(* CODESYS project shid.project

Project tree, tasks and I/O mapping:
  Device : CECC-LK, Festo AG & Co. KG, order no. 574418, version 3.5.7.27
    application Application
      libraries: Standard, * (System); CAA CiA 405, 3.5.0.0 (CAA Technical Workgroup); Solution Center Library, 3.5.8.0 (Festo Didactic SE - Customer Solution Center); OPAK_RFID, 3.5.0.0 (elrest Automationssysteme GmbH); CAA DTUtil Extern, * (CAA Technical Workgroup)
      task MainTask (cyclic, interval t#20ms, priority 20) calls PLC_TO_PC_PROJECT_PRG
      program PLC_PRG [ST]
      program RFID_PRG [ST]
      global variables IO
      program timer_PRG [ST]
      program customTimer_PRG [ST]
      program TCP_PRG [ST]
      program PLC_TO_PC_PROJECT_PRG [ST]
    Onboard : CECC 14I/8O, Festo AG & Co. KG, version 3.4.5.5
        unmapped channels: Onboard Input, Onboard Output
      Digital Inputs
          unmapped channels: Onboard Input
      Digital Outputs
          unmapped channels: Onboard Output
    CAN : CANbus, 3S - Smart Software Solutions GmbH, version 3.5.10.0
        settings: Baudrate = 1000
      CANopen : CANopen_Manager, 3S - Smart Software Solutions GmbH, version 3.5.10.0
          settings: Sync CycleTime in Microseconds = 8000; Synchronous Window Length = 0; Enable Heartbeat generation = FALSE; Factory Settings Default = FALSE; Expert Settings Default = TRUE; ConfigVersion = 50659584
        BL20_GWBR_CANOPEN : BL20-GWBR-CANOPEN, TURCK, order no. 6827167, version Revision=16#00040017, FileVersion=4.23
            settings: General Options.Reset Node = FALSE; NODEIDSAVED = 2; SDO Timeout = 1000000; PDO_Autoconfig = TRUE; EXPERTSETTINGS = TRUE; Emergency-General Parameters.Emergency COBID = 16#00000082; Settings.COBID = 16#00000202; Settings.Transmission Type = 16#FF; Settings.available PDO-Parameter.Inhibit Time available = FALSE; Settings.available PDO-Parameter.Event Timer available = FALSE; Settings.Inhibit Time = 0; Settings.Event Timer = 0; Generic COBID = '$NODEID+16#0200'; Process by CANopenManager = TRUE; Settings.COBID = 16#00000302; Settings.Transmission Type = 16#FF; Settings.available PDO-Parameter.Inhibit Time available = FALSE; Settings.available PDO-Parameter.Event Timer available = FALSE; Settings.Inhibit Time = 0; Settings.Event Timer = 0; Generic COBID = '$NODEID+16#0300'; Process by CANopenManager = TRUE; Settings.COBID = 16#00000182; Settings.Transmission Type = 16#FF; Settings.available PDO-Parameter.Inhibit Time available = TRUE; Settings.available PDO-Parameter.Event Timer available = TRUE; Settings.Inhibit Time = 0; Settings.Event Timer = 0; Generic COBID = '$NODEID+16#0180'; Process by CANopenManager = TRUE; Settings.COBID = 16#00000282; Settings.Transmission Type = 16#FF; Settings.available PDO-Parameter.Inhibit Time available = TRUE; Settings.available PDO-Parameter.Event Timer available = TRUE; Settings.Inhibit Time = 0; Settings.Event Timer = 0; Generic COBID = '$NODEID+16#0280'; Process by CANopenManager = TRUE; WriteOutput8Bit : Generic_BL20_4DO.Index = 16#6200; WriteOutput8Bit : Generic_BL20_4DO.Subindex = 16#01;
              WriteOutput8Bit : Generic_BL20_4DO.ObjectLength = 8; WriteOutput8Bit : Generic_BL20_4DO_2.Index = 16#6200; WriteOutput8Bit : Generic_BL20_4DO_2.Subindex = 16#02; WriteOutput8Bit : Generic_BL20_4DO_2.ObjectLength = 8; WriteAnalogueOutput16 : Generic_BL20_2AO.Index = 16#6411; WriteAnalogueOutput16 : Generic_BL20_2AO.Subindex = 16#01; WriteAnalogueOutput16 : Generic_BL20_2AO.ObjectLength = 16; WriteAnalogueOutput16 : Generic_BL20_2AO.Index = 16#6411; WriteAnalogueOutput16 : Generic_BL20_2AO.Subindex = 16#02; WriteAnalogueOutput16 : Generic_BL20_2AO.ObjectLength = 16; ReadInput8Bit : Generic_BL20_4DI.Index = 16#6000; ReadInput8Bit : Generic_BL20_4DI.Subindex = 16#01; ReadInput8Bit : Generic_BL20_4DI.ObjectLength = 8; ReadAnalogueInput16Bit : Generic_BL20_4AI.Index = 16#6401; ReadAnalogueInput16Bit : Generic_BL20_4AI.Subindex = 16#01; ReadAnalogueInput16Bit : Generic_BL20_4AI.ObjectLength = 16; ReadAnalogueInput16Bit : Generic_BL20_4AI.Index = 16#6401; ReadAnalogueInput16Bit : Generic_BL20_4AI.Subindex = 16#02; ReadAnalogueInput16Bit : Generic_BL20_4AI.ObjectLength = 16; ReadAnalogueInput16Bit : Generic_BL20_4AI.Index = 16#6401; ReadAnalogueInput16Bit : Generic_BL20_4AI.Subindex = 16#03; ReadAnalogueInput16Bit : Generic_BL20_4AI.ObjectLength = 16; ReadAnalogueInput16Bit : Generic_BL20_4AI.Index = 16#6401; ReadAnalogueInput16Bit : Generic_BL20_4AI.Subindex = 16#04; ReadAnalogueInput16Bit : Generic_BL20_4AI.ObjectLength = 16; SDO List.Set Guardtime.Index = 16#100C; SDO List.Set Guardtime.Subindex = 16#00; SDO List.Set Guardtime.Value = 16#00000000; SDO List.Set Guardtime.Size = 16; SDO List.Set Guardtime.AbortIfError = FALSE; SDO List.Set Guardtime.JumpToLine = FALSE; SDO List.Set Guardtime.Line = 0; SDO List.Set Lifetime.Index = 16#100D; SDO List.Set Lifetime.Subindex = 16#00; SDO List.Set Lifetime.Value = 16#00000000; SDO List.Set Lifetime.Size = 8; SDO List.Set Lifetime.AbortIfError = FALSE; SDO List.Set Lifetime.JumpToLine = FALSE; SDO List.Set Lifetime.Line = 0; SDO List.Disable Emcy CobID.Index = 16#1014;
              SDO List.Disable Emcy CobID.Subindex = 16#00; SDO List.Disable Emcy CobID.Value = 16#80000082; SDO List.Disable Emcy CobID.Size = 32; SDO List.Disable Emcy CobID.AbortIfError = FALSE; SDO List.Disable Emcy CobID.JumpToLine = FALSE; SDO List.Disable Emcy CobID.Line = 0; SDO List.Set Emcy CobID.Index = 16#1014; SDO List.Set Emcy CobID.Subindex = 16#00; SDO List.Set Emcy CobID.Value = 16#00000082; SDO List.Set Emcy CobID.Size = 32; SDO List.Set Emcy CobID.AbortIfError = FALSE; SDO List.Set Emcy CobID.JumpToLine = FALSE; SDO List.Set Emcy CobID.Line = 0; SDO List.Set Heartbeat Consumer.Index = 16#1016; SDO List.Set Heartbeat Consumer.Subindex = 16#01; SDO List.Set Heartbeat Consumer.Value = 0; SDO List.Set Heartbeat Consumer.Size = 32; SDO List.Set Heartbeat Consumer.AbortIfError = FALSE; SDO List.Set Heartbeat Consumer.JumpToLine = FALSE; SDO List.Set Heartbeat Consumer.Line = 0; SDO List.Set Heartbeat Producer.Index = 16#1017; SDO List.Set Heartbeat Producer.Subindex = 16#00; SDO List.Set Heartbeat Producer.Value = 16#00000000; SDO List.Set Heartbeat Producer.Size = 16; SDO List.Set Heartbeat Producer.AbortIfError = FALSE; SDO List.Set Heartbeat Producer.JumpToLine = FALSE; SDO List.Set Heartbeat Producer.Line = 0; SDO List.Disable PDO.Index = 16#1400; SDO List.Disable PDO.Subindex = 16#01; SDO List.Disable PDO.Value = 16#80000202; SDO List.Disable PDO.Size = 32; SDO List.Disable PDO.AbortIfError = FALSE; SDO List.Disable PDO.JumpToLine = FALSE; SDO List.Disable PDO.Line = 0; SDO List.Set transmission type.Index = 16#1400; SDO List.Set transmission type.Subindex = 16#02; SDO List.Set transmission type.Value = 16#FF; SDO List.Set transmission type.Size = 8; SDO List.Set transmission type.AbortIfError = FALSE; SDO List.Set transmission type.JumpToLine = FALSE;
              SDO List.Set transmission type.Line = 0; SDO List.Clear pdo mapping.Index = 16#1600; SDO List.Clear pdo mapping.Subindex = 16#00; SDO List.Clear pdo mapping.Value = 16#0; SDO List.Clear pdo mapping.Size = 8; SDO List.Clear pdo mapping.AbortIfError = FALSE; SDO List.Clear pdo mapping.JumpToLine = FALSE; SDO List.Clear pdo mapping.Line = 0; SDO List.Set Mapping.Index = 16#1600; SDO List.Set Mapping.Subindex = 16#01; SDO List.Set Mapping.Value = 16#62000108; SDO List.Set Mapping.Size = 32; SDO List.Set Mapping.AbortIfError = FALSE; SDO List.Set Mapping.JumpToLine = FALSE; SDO List.Set Mapping.Line = 0; SDO List.Set Mapping.Index = 16#1600; SDO List.Set Mapping.Subindex = 16#02; SDO List.Set Mapping.Value = 16#62000208; SDO List.Set Mapping.Size = 32; SDO List.Set Mapping.AbortIfError = FALSE; SDO List.Set Mapping.JumpToLine = FALSE; SDO List.Set Mapping.Line = 0; SDO List.Set number of mappings.Index = 16#1600; SDO List.Set number of mappings.Subindex = 16#00; SDO List.Set number of mappings.Value = 16#02; SDO List.Set number of mappings.Size = 8; SDO List.Set number of mappings.AbortIfError = FALSE; SDO List.Set number of mappings.JumpToLine = FALSE; SDO List.Set number of mappings.Line = 0; SDO List.Set and enable COB-ID.Index = 16#1400; SDO List.Set and enable COB-ID.Subindex = 16#01; SDO List.Set and enable COB-ID.Value = 16#00000202; SDO List.Set and enable COB-ID.Size = 32; SDO List.Set and enable COB-ID.AbortIfError = FALSE; SDO List.Set and enable COB-ID.JumpToLine = FALSE; SDO List.Set and enable COB-ID.Line = 0; SDO List.Disable PDO.Index = 16#1401; SDO List.Disable PDO.Subindex = 16#01; SDO List.Disable PDO.Value = 16#80000302; SDO List.Disable PDO.Size = 32;
              SDO List.Disable PDO.AbortIfError = FALSE; SDO List.Disable PDO.JumpToLine = FALSE; SDO List.Disable PDO.Line = 0; SDO List.Set transmission type.Index = 16#1401; SDO List.Set transmission type.Subindex = 16#02; SDO List.Set transmission type.Value = 16#FF; SDO List.Set transmission type.Size = 8; SDO List.Set transmission type.AbortIfError = FALSE; SDO List.Set transmission type.JumpToLine = FALSE; SDO List.Set transmission type.Line = 0; SDO List.Clear pdo mapping.Index = 16#1601; SDO List.Clear pdo mapping.Subindex = 16#00; SDO List.Clear pdo mapping.Value = 16#0; SDO List.Clear pdo mapping.Size = 8; SDO List.Clear pdo mapping.AbortIfError = FALSE; SDO List.Clear pdo mapping.JumpToLine = FALSE; SDO List.Clear pdo mapping.Line = 0; SDO List.Set Mapping.Index = 16#1601; SDO List.Set Mapping.Subindex = 16#01; SDO List.Set Mapping.Value = 16#64110110; SDO List.Set Mapping.Size = 32; SDO List.Set Mapping.AbortIfError = FALSE; SDO List.Set Mapping.JumpToLine = FALSE; SDO List.Set Mapping.Line = 0; SDO List.Set Mapping.Index = 16#1601; SDO List.Set Mapping.Subindex = 16#02; SDO List.Set Mapping.Value = 16#64110210; SDO List.Set Mapping.Size = 32; SDO List.Set Mapping.AbortIfError = FALSE; SDO List.Set Mapping.JumpToLine = FALSE; SDO List.Set Mapping.Line = 0; SDO List.Set number of mappings.Index = 16#1601; SDO List.Set number of mappings.Subindex = 16#00; SDO List.Set number of mappings.Value = 16#02; SDO List.Set number of mappings.Size = 8; SDO List.Set number of mappings.AbortIfError = FALSE; SDO List.Set number of mappings.JumpToLine = FALSE; SDO List.Set number of mappings.Line = 0; SDO List.Set and enable COB-ID.Index = 16#1401; SDO List.Set and enable COB-ID.Subindex = 16#01;
              SDO List.Set and enable COB-ID.Value = 16#00000302; SDO List.Set and enable COB-ID.Size = 32; SDO List.Set and enable COB-ID.AbortIfError = FALSE; SDO List.Set and enable COB-ID.JumpToLine = FALSE; SDO List.Set and enable COB-ID.Line = 0; SDO List.Disable PDO.Index = 16#1800; SDO List.Disable PDO.Subindex = 16#01; SDO List.Disable PDO.Value = 16#80000182; SDO List.Disable PDO.Size = 32; SDO List.Disable PDO.AbortIfError = FALSE; SDO List.Disable PDO.JumpToLine = FALSE; SDO List.Disable PDO.Line = 0; SDO List.Set transmission type.Index = 16#1800; SDO List.Set transmission type.Subindex = 16#02; SDO List.Set transmission type.Value = 16#FF; SDO List.Set transmission type.Size = 8; SDO List.Set transmission type.AbortIfError = FALSE; SDO List.Set transmission type.JumpToLine = FALSE; SDO List.Set transmission type.Line = 0; SDO List.Set inhibit time.Index = 16#1800; SDO List.Set inhibit time.Subindex = 16#03; SDO List.Set inhibit time.Value = 16#0000; SDO List.Set inhibit time.Size = 16; SDO List.Set inhibit time.AbortIfError = FALSE; SDO List.Set inhibit time.JumpToLine = FALSE; SDO List.Set inhibit time.Line = 0; SDO List.Set event time.Index = 16#1800; SDO List.Set event time.Subindex = 16#05; SDO List.Set event time.Value = 16#0000; SDO List.Set event time.Size = 16; SDO List.Set event time.AbortIfError = FALSE; SDO List.Set event time.JumpToLine = FALSE; SDO List.Set event time.Line = 0; SDO List.Clear pdo mapping.Index = 16#1A00; SDO List.Clear pdo mapping.Subindex = 16#00; SDO List.Clear pdo mapping.Value = 16#0; SDO List.Clear pdo mapping.Size = 8; SDO List.Clear pdo mapping.AbortIfError = FALSE; SDO List.Clear pdo mapping.JumpToLine = FALSE; SDO List.Clear pdo mapping.Line = 0;
              SDO List.Set Mapping.Index = 16#1A00; SDO List.Set Mapping.Subindex = 16#01; SDO List.Set Mapping.Value = 16#60000108; SDO List.Set Mapping.Size = 32; SDO List.Set Mapping.AbortIfError = FALSE; SDO List.Set Mapping.JumpToLine = FALSE; SDO List.Set Mapping.Line = 0; SDO List.Set number of mappings.Index = 16#1A00; SDO List.Set number of mappings.Subindex = 16#00; SDO List.Set number of mappings.Value = 16#01; SDO List.Set number of mappings.Size = 8; SDO List.Set number of mappings.AbortIfError = FALSE; SDO List.Set number of mappings.JumpToLine = FALSE; SDO List.Set number of mappings.Line = 0; SDO List.Set and enable COB-ID.Index = 16#1800; SDO List.Set and enable COB-ID.Subindex = 16#01; SDO List.Set and enable COB-ID.Value = 16#00000182; SDO List.Set and enable COB-ID.Size = 32; SDO List.Set and enable COB-ID.AbortIfError = FALSE; SDO List.Set and enable COB-ID.JumpToLine = FALSE; SDO List.Set and enable COB-ID.Line = 0; SDO List.Disable PDO.Index = 16#1801; SDO List.Disable PDO.Subindex = 16#01; SDO List.Disable PDO.Value = 16#80000282; SDO List.Disable PDO.Size = 32; SDO List.Disable PDO.AbortIfError = FALSE; SDO List.Disable PDO.JumpToLine = FALSE; SDO List.Disable PDO.Line = 0; SDO List.Set transmission type.Index = 16#1801; SDO List.Set transmission type.Subindex = 16#02; SDO List.Set transmission type.Value = 16#FF; SDO List.Set transmission type.Size = 8; SDO List.Set transmission type.AbortIfError = FALSE; SDO List.Set transmission type.JumpToLine = FALSE; SDO List.Set transmission type.Line = 0; SDO List.Set inhibit time.Index = 16#1801; SDO List.Set inhibit time.Subindex = 16#03; SDO List.Set inhibit time.Value = 16#0000; SDO List.Set inhibit time.Size = 16; SDO List.Set inhibit time.AbortIfError = FALSE;
              SDO List.Set inhibit time.JumpToLine = FALSE; SDO List.Set inhibit time.Line = 0; SDO List.Set event time.Index = 16#1801; SDO List.Set event time.Subindex = 16#05; SDO List.Set event time.Value = 16#0000; SDO List.Set event time.Size = 16; SDO List.Set event time.AbortIfError = FALSE; SDO List.Set event time.JumpToLine = FALSE; SDO List.Set event time.Line = 0; SDO List.Clear pdo mapping.Index = 16#1A01; SDO List.Clear pdo mapping.Subindex = 16#00; SDO List.Clear pdo mapping.Value = 16#0; SDO List.Clear pdo mapping.Size = 8; SDO List.Clear pdo mapping.AbortIfError = FALSE; SDO List.Clear pdo mapping.JumpToLine = FALSE; SDO List.Clear pdo mapping.Line = 0; SDO List.Set Mapping.Index = 16#1A01; SDO List.Set Mapping.Subindex = 16#01; SDO List.Set Mapping.Value = 16#64010110; SDO List.Set Mapping.Size = 32; SDO List.Set Mapping.AbortIfError = FALSE; SDO List.Set Mapping.JumpToLine = FALSE; SDO List.Set Mapping.Line = 0; SDO List.Set Mapping.Index = 16#1A01; SDO List.Set Mapping.Subindex = 16#02; SDO List.Set Mapping.Value = 16#64010210; SDO List.Set Mapping.Size = 32; SDO List.Set Mapping.AbortIfError = FALSE; SDO List.Set Mapping.JumpToLine = FALSE; SDO List.Set Mapping.Line = 0; SDO List.Set Mapping.Index = 16#1A01; SDO List.Set Mapping.Subindex = 16#03; SDO List.Set Mapping.Value = 16#64010310; SDO List.Set Mapping.Size = 32; SDO List.Set Mapping.AbortIfError = FALSE; SDO List.Set Mapping.JumpToLine = FALSE; SDO List.Set Mapping.Line = 0; SDO List.Set Mapping.Index = 16#1A01; SDO List.Set Mapping.Subindex = 16#04; SDO List.Set Mapping.Value = 16#64010410;
              SDO List.Set Mapping.Size = 32; SDO List.Set Mapping.AbortIfError = FALSE; SDO List.Set Mapping.JumpToLine = FALSE; SDO List.Set Mapping.Line = 0; SDO List.Set number of mappings.Index = 16#1A01; SDO List.Set number of mappings.Subindex = 16#00; SDO List.Set number of mappings.Value = 16#04; SDO List.Set number of mappings.Size = 8; SDO List.Set number of mappings.AbortIfError = FALSE; SDO List.Set number of mappings.JumpToLine = FALSE; SDO List.Set number of mappings.Line = 0; SDO List.Set and enable COB-ID.Index = 16#1801; SDO List.Set and enable COB-ID.Subindex = 16#01; SDO List.Set and enable COB-ID.Value = 16#00000282; SDO List.Set and enable COB-ID.Size = 32; SDO List.Set and enable COB-ID.AbortIfError = FALSE; SDO List.Set and enable COB-ID.JumpToLine = FALSE; SDO List.Set and enable COB-ID.Line = 0; ConfigVersion = 50659584
          Generic_BL20_4DI : Generic BL20-4DI, TURCK, order no. 0, version Revision=16#00040017, FileVersion=4.23
              settings: Number of Params = 1; ReadInput8Bit : Generic_BL20_4DI.Index = 16#6000; ReadInput8Bit : Generic_BL20_4DI.Subindex = 16#01; ReadInput8Bit : Generic_BL20_4DI.Startbit = 0; ReadInput8Bit : Generic_BL20_4DI.Endbit = 3
              unmapped channels: ReadInput8Bit : Generic_BL20_4DI
          Generic_BL20_4DI_1 : Generic BL20-4DI, TURCK, order no. 0, version Revision=16#00040017, FileVersion=4.23
              settings: Number of Params = 1; ReadInput8Bit : Generic_BL20_4DI.Index = 16#6000; ReadInput8Bit : Generic_BL20_4DI.Subindex = 16#01; ReadInput8Bit : Generic_BL20_4DI.Startbit = 4; ReadInput8Bit : Generic_BL20_4DI.Endbit = 7
              unmapped channels: ReadInput8Bit : Generic_BL20_4DI
          Generic_BL20_BR_PF : Generic BL20-BR/-PF, TURCK, order no. 0, version Revision=16#00040017, FileVersion=4.23
          Generic_BL20_4DO : Generic BL20-4DO, TURCK, order no. 0, version Revision=16#00040017, FileVersion=4.23
              settings: Number of Params = 1; WriteOutput8Bit : Generic_BL20_4DO.Index = 16#6200; WriteOutput8Bit : Generic_BL20_4DO.Subindex = 16#01; WriteOutput8Bit : Generic_BL20_4DO.Startbit = 0; WriteOutput8Bit : Generic_BL20_4DO.Endbit = 3
              unmapped channels: WriteOutput8Bit : Generic_BL20_4DO
          Generic_BL20_4DO_1 : Generic BL20-4DO, TURCK, order no. 0, version Revision=16#00040017, FileVersion=4.23
              settings: Number of Params = 1; WriteOutput8Bit : Generic_BL20_4DO.Index = 16#6200; WriteOutput8Bit : Generic_BL20_4DO.Subindex = 16#01; WriteOutput8Bit : Generic_BL20_4DO.Startbit = 4; WriteOutput8Bit : Generic_BL20_4DO.Endbit = 7
              unmapped channels: WriteOutput8Bit : Generic_BL20_4DO
          Generic_BL20_4DO_2 : Generic BL20-4DO, TURCK, order no. 0, version Revision=16#00040017, FileVersion=4.23
              settings: Number of Params = 1; WriteOutput8Bit : Generic_BL20_4DO_2.Index = 16#6200; WriteOutput8Bit : Generic_BL20_4DO_2.Subindex = 16#02; WriteOutput8Bit : Generic_BL20_4DO_2.Startbit = 0; WriteOutput8Bit : Generic_BL20_4DO_2.Endbit = 3
              unmapped channels: WriteOutput8Bit : Generic_BL20_4DO_2
          Generic_BL20_4DO_3 : Generic BL20-4DO, TURCK, order no. 0, version Revision=16#00040017, FileVersion=4.23
              settings: Number of Params = 1; WriteOutput8Bit : Generic_BL20_4DO_2.Index = 16#6200; WriteOutput8Bit : Generic_BL20_4DO_2.Subindex = 16#02; WriteOutput8Bit : Generic_BL20_4DO_2.Startbit = 4; WriteOutput8Bit : Generic_BL20_4DO_2.Endbit = 7
              unmapped channels: WriteOutput8Bit : Generic_BL20_4DO_2
          Generic_BL20_4AI : Generic BL20-4AI, TURCK, order no. 0, version Revision=16#00040017, FileVersion=4.23
              settings: Number of Params = 4; ReadAnalogueInput16Bit : Generic_BL20_4AI.Index = 16#6401; ReadAnalogueInput16Bit : Generic_BL20_4AI.Subindex = 16#01; ReadAnalogueInput16Bit : Generic_BL20_4AI.Startbit = 0; ReadAnalogueInput16Bit : Generic_BL20_4AI.Endbit = 15; ReadAnalogueInput16Bit : Generic_BL20_4AI.Index = 16#6401; ReadAnalogueInput16Bit : Generic_BL20_4AI.Subindex = 16#02; ReadAnalogueInput16Bit : Generic_BL20_4AI.Startbit = 0; ReadAnalogueInput16Bit : Generic_BL20_4AI.Endbit = 15; ReadAnalogueInput16Bit : Generic_BL20_4AI.Index = 16#6401; ReadAnalogueInput16Bit : Generic_BL20_4AI.Subindex = 16#03; ReadAnalogueInput16Bit : Generic_BL20_4AI.Startbit = 0; ReadAnalogueInput16Bit : Generic_BL20_4AI.Endbit = 15; ReadAnalogueInput16Bit : Generic_BL20_4AI.Index = 16#6401; ReadAnalogueInput16Bit : Generic_BL20_4AI.Subindex = 16#04; ReadAnalogueInput16Bit : Generic_BL20_4AI.Startbit = 0; ReadAnalogueInput16Bit : Generic_BL20_4AI.Endbit = 15
              unmapped channels: ReadAnalogueInput16Bit : Generic_BL20_4AI, ReadAnalogueInput16Bit : Generic_BL20_4AI, ReadAnalogueInput16Bit : Generic_BL20_4AI, ReadAnalogueInput16Bit : Generic_BL20_4AI
          Generic_BL20_2AO : Generic BL20-2AO, TURCK, order no. 0, version Revision=16#00040017, FileVersion=4.23
              settings: Number of Params = 2; WriteAnalogueOutput16 : Generic_BL20_2AO.Index = 16#6411; WriteAnalogueOutput16 : Generic_BL20_2AO.Subindex = 16#01; WriteAnalogueOutput16 : Generic_BL20_2AO.Startbit = 0; WriteAnalogueOutput16 : Generic_BL20_2AO.Endbit = 15; WriteAnalogueOutput16 : Generic_BL20_2AO.Index = 16#6411; WriteAnalogueOutput16 : Generic_BL20_2AO.Subindex = 16#02; WriteAnalogueOutput16 : Generic_BL20_2AO.Startbit = 0; WriteAnalogueOutput16 : Generic_BL20_2AO.Endbit = 15
              unmapped channels: WriteAnalogueOutput16 : Generic_BL20_2AO, WriteAnalogueOutput16 : Generic_BL20_2AO
        DTM425 : DTM425, ifm electronic gmbh, order no. DTM425, version Revision=16#00000000, FileVersion=8.2, File=DTM425.eds
            settings: General Options.Reset Node = FALSE; NODEIDSAVED = 32; SDO Timeout = 1000000; PDO_Autoconfig = FALSE; EXPERTSETTINGS = TRUE; Emergency-General Parameters.Emergency COBID = 16#000000A0; PDO 16#1400.COBID = 16#00000220; Process by CANopenManager = TRUE; PDO 16#1401.COBID = 16#00000320; Process by CANopenManager = TRUE; PDO 16#1402.COBID = 16#00000420; Process by CANopenManager = TRUE; PDO 16#1403.COBID = 16#00000520; Process by CANopenManager = TRUE; PDO 16#1800.COBID = 16#000001A0; PDO 16#1800.Event Timer = 0; Process by CANopenManager = TRUE; PDO 16#1801.COBID = 16#000002A0; PDO 16#1801.Event Timer = 0; Process by CANopenManager = TRUE; PDO 16#1802.COBID = 16#000003A0; PDO 16#1802.Event Timer = 0; Process by CANopenManager = TRUE; PDO 16#1803.COBID = 16#000004A0; PDO 16#1803.Event Timer = 0; Process by CANopenManager = TRUE; Write Data (mappable): Write Trigger.Subindex = 16#00; Write Data (mappable): Data_sub1.Subindex = 16#01; Write Data (mappable): Data_sub2.Subindex = 16#02; Write Data (mappable): Data_sub3.Subindex = 16#03; Device Status.Subindex = 16#00; Read Data (mappable): Data_sub1.Subindex = 16#01; Read Data (mappable): Data_sub2.Subindex = 16#02; Read Data (mappable): Data_sub3.Subindex = 16#03; SDO List.Disable Emcy CobID.Index = 16#1014; SDO List.Disable Emcy CobID.Subindex = 16#00; SDO List.Disable Emcy CobID.Value = 16#800000A0; SDO List.Disable Emcy CobID.Size = 32; SDO List.Disable Emcy CobID.AbortIfError = FALSE; SDO List.Disable Emcy CobID.JumpToLine = FALSE;
              SDO List.Disable Emcy CobID.Line = 0; SDO List.Set Emcy CobID.Index = 16#1014; SDO List.Set Emcy CobID.Subindex = 16#00; SDO List.Set Emcy CobID.Value = 16#000000A0; SDO List.Set Emcy CobID.Size = 32; SDO List.Set Emcy CobID.AbortIfError = FALSE; SDO List.Set Emcy CobID.JumpToLine = FALSE; SDO List.Set Emcy CobID.Line = 0; SDO List.Set Heartbeat Producer.Index = 16#1017; SDO List.Set Heartbeat Producer.Subindex = 16#00; SDO List.Set Heartbeat Producer.Value = 16#00000000; SDO List.Set Heartbeat Producer.Size = 16; SDO List.Set Heartbeat Producer.AbortIfError = FALSE; SDO List.Set Heartbeat Producer.JumpToLine = FALSE; SDO List.Set Heartbeat Producer.Line = 0; SDO List.Disable PDO.Index = 16#1400; SDO List.Disable PDO.Subindex = 16#01; SDO List.Disable PDO.Value = 16#80000220; SDO List.Disable PDO.Size = 32; SDO List.Disable PDO.AbortIfError = FALSE; SDO List.Disable PDO.JumpToLine = FALSE; SDO List.Disable PDO.Line = 0; SDO List.Set transmission type.Index = 16#1400; SDO List.Set transmission type.Subindex = 16#02; SDO List.Set transmission type.Value = 16#FF; SDO List.Set transmission type.Size = 8; SDO List.Set transmission type.AbortIfError = FALSE; SDO List.Set transmission type.JumpToLine = FALSE; SDO List.Set transmission type.Line = 0; SDO List.Clear pdo mapping.Index = 16#1600; SDO List.Clear pdo mapping.Subindex = 16#00; SDO List.Clear pdo mapping.Value = 16#0; SDO List.Clear pdo mapping.Size = 8; SDO List.Clear pdo mapping.AbortIfError = FALSE; SDO List.Clear pdo mapping.JumpToLine = FALSE; SDO List.Clear pdo mapping.Line = 0; SDO List.Set Mapping.Index = 16#1600; SDO List.Set Mapping.Subindex = 16#01; SDO List.Set Mapping.Value = 16#230F0040; SDO List.Set Mapping.Size = 32;
              SDO List.Set Mapping.AbortIfError = FALSE; SDO List.Set Mapping.JumpToLine = FALSE; SDO List.Set Mapping.Line = 0; SDO List.Set number of mappings.Index = 16#1600; SDO List.Set number of mappings.Subindex = 16#00; SDO List.Set number of mappings.Value = 16#01; SDO List.Set number of mappings.Size = 8; SDO List.Set number of mappings.AbortIfError = FALSE; SDO List.Set number of mappings.JumpToLine = FALSE; SDO List.Set number of mappings.Line = 0; SDO List.Set and enable COB-ID.Index = 16#1400; SDO List.Set and enable COB-ID.Subindex = 16#01; SDO List.Set and enable COB-ID.Value = 16#00000220; SDO List.Set and enable COB-ID.Size = 32; SDO List.Set and enable COB-ID.AbortIfError = FALSE; SDO List.Set and enable COB-ID.JumpToLine = FALSE; SDO List.Set and enable COB-ID.Line = 0; SDO List.Disable PDO.Index = 16#1401; SDO List.Disable PDO.Subindex = 16#01; SDO List.Disable PDO.Value = 16#80000320; SDO List.Disable PDO.Size = 32; SDO List.Disable PDO.AbortIfError = FALSE; SDO List.Disable PDO.JumpToLine = FALSE; SDO List.Disable PDO.Line = 0; SDO List.Set transmission type.Index = 16#1401; SDO List.Set transmission type.Subindex = 16#02; SDO List.Set transmission type.Value = 16#FF; SDO List.Set transmission type.Size = 8; SDO List.Set transmission type.AbortIfError = FALSE; SDO List.Set transmission type.JumpToLine = FALSE; SDO List.Set transmission type.Line = 0; SDO List.Clear pdo mapping.Index = 16#1601; SDO List.Clear pdo mapping.Subindex = 16#00; SDO List.Clear pdo mapping.Value = 16#0; SDO List.Clear pdo mapping.Size = 8; SDO List.Clear pdo mapping.AbortIfError = FALSE; SDO List.Clear pdo mapping.JumpToLine = FALSE; SDO List.Clear pdo mapping.Line = 0; SDO List.Set Mapping.Index = 16#1601; SDO List.Set Mapping.Subindex = 16#01;
              SDO List.Set Mapping.Value = 16#230A0140; SDO List.Set Mapping.Size = 32; SDO List.Set Mapping.AbortIfError = FALSE; SDO List.Set Mapping.JumpToLine = FALSE; SDO List.Set Mapping.Line = 0; SDO List.Set number of mappings.Index = 16#1601; SDO List.Set number of mappings.Subindex = 16#00; SDO List.Set number of mappings.Value = 16#01; SDO List.Set number of mappings.Size = 8; SDO List.Set number of mappings.AbortIfError = FALSE; SDO List.Set number of mappings.JumpToLine = FALSE; SDO List.Set number of mappings.Line = 0; SDO List.Set and enable COB-ID.Index = 16#1401; SDO List.Set and enable COB-ID.Subindex = 16#01; SDO List.Set and enable COB-ID.Value = 16#00000320; SDO List.Set and enable COB-ID.Size = 32; SDO List.Set and enable COB-ID.AbortIfError = FALSE; SDO List.Set and enable COB-ID.JumpToLine = FALSE; SDO List.Set and enable COB-ID.Line = 0; SDO List.Disable PDO.Index = 16#1402; SDO List.Disable PDO.Subindex = 16#01; SDO List.Disable PDO.Value = 16#80000420; SDO List.Disable PDO.Size = 32; SDO List.Disable PDO.AbortIfError = FALSE; SDO List.Disable PDO.JumpToLine = FALSE; SDO List.Disable PDO.Line = 0; SDO List.Set transmission type.Index = 16#1402; SDO List.Set transmission type.Subindex = 16#02; SDO List.Set transmission type.Value = 16#FF; SDO List.Set transmission type.Size = 8; SDO List.Set transmission type.AbortIfError = FALSE; SDO List.Set transmission type.JumpToLine = FALSE; SDO List.Set transmission type.Line = 0; SDO List.Clear pdo mapping.Index = 16#1602; SDO List.Clear pdo mapping.Subindex = 16#00; SDO List.Clear pdo mapping.Value = 16#0; SDO List.Clear pdo mapping.Size = 8; SDO List.Clear pdo mapping.AbortIfError = FALSE; SDO List.Clear pdo mapping.JumpToLine = FALSE; SDO List.Clear pdo mapping.Line = 0;
              SDO List.Set Mapping.Index = 16#1602; SDO List.Set Mapping.Subindex = 16#01; SDO List.Set Mapping.Value = 16#230A0240; SDO List.Set Mapping.Size = 32; SDO List.Set Mapping.AbortIfError = FALSE; SDO List.Set Mapping.JumpToLine = FALSE; SDO List.Set Mapping.Line = 0; SDO List.Set number of mappings.Index = 16#1602; SDO List.Set number of mappings.Subindex = 16#00; SDO List.Set number of mappings.Value = 16#01; SDO List.Set number of mappings.Size = 8; SDO List.Set number of mappings.AbortIfError = FALSE; SDO List.Set number of mappings.JumpToLine = FALSE; SDO List.Set number of mappings.Line = 0; SDO List.Set and enable COB-ID.Index = 16#1402; SDO List.Set and enable COB-ID.Subindex = 16#01; SDO List.Set and enable COB-ID.Value = 16#00000420; SDO List.Set and enable COB-ID.Size = 32; SDO List.Set and enable COB-ID.AbortIfError = FALSE; SDO List.Set and enable COB-ID.JumpToLine = FALSE; SDO List.Set and enable COB-ID.Line = 0; SDO List.Disable PDO.Index = 16#1403; SDO List.Disable PDO.Subindex = 16#01; SDO List.Disable PDO.Value = 16#80000520; SDO List.Disable PDO.Size = 32; SDO List.Disable PDO.AbortIfError = FALSE; SDO List.Disable PDO.JumpToLine = FALSE; SDO List.Disable PDO.Line = 0; SDO List.Set transmission type.Index = 16#1403; SDO List.Set transmission type.Subindex = 16#02; SDO List.Set transmission type.Value = 16#FF; SDO List.Set transmission type.Size = 8; SDO List.Set transmission type.AbortIfError = FALSE; SDO List.Set transmission type.JumpToLine = FALSE; SDO List.Set transmission type.Line = 0; SDO List.Clear pdo mapping.Index = 16#1603; SDO List.Clear pdo mapping.Subindex = 16#00; SDO List.Clear pdo mapping.Value = 16#0; SDO List.Clear pdo mapping.Size = 8; SDO List.Clear pdo mapping.AbortIfError = FALSE;
              SDO List.Clear pdo mapping.JumpToLine = FALSE; SDO List.Clear pdo mapping.Line = 0; SDO List.Set Mapping.Index = 16#1603; SDO List.Set Mapping.Subindex = 16#01; SDO List.Set Mapping.Value = 16#230A0340; SDO List.Set Mapping.Size = 32; SDO List.Set Mapping.AbortIfError = FALSE; SDO List.Set Mapping.JumpToLine = FALSE; SDO List.Set Mapping.Line = 0; SDO List.Set number of mappings.Index = 16#1603; SDO List.Set number of mappings.Subindex = 16#00; SDO List.Set number of mappings.Value = 16#01; SDO List.Set number of mappings.Size = 8; SDO List.Set number of mappings.AbortIfError = FALSE; SDO List.Set number of mappings.JumpToLine = FALSE; SDO List.Set number of mappings.Line = 0; SDO List.Set and enable COB-ID.Index = 16#1403; SDO List.Set and enable COB-ID.Subindex = 16#01; SDO List.Set and enable COB-ID.Value = 16#00000520; SDO List.Set and enable COB-ID.Size = 32; SDO List.Set and enable COB-ID.AbortIfError = FALSE; SDO List.Set and enable COB-ID.JumpToLine = FALSE; SDO List.Set and enable COB-ID.Line = 0; SDO List.Disable PDO.Index = 16#1800; SDO List.Disable PDO.Subindex = 16#01; SDO List.Disable PDO.Value = 16#800001A0; SDO List.Disable PDO.Size = 32; SDO List.Disable PDO.AbortIfError = FALSE; SDO List.Disable PDO.JumpToLine = FALSE; SDO List.Disable PDO.Line = 0; SDO List.Set transmission type.Index = 16#1800; SDO List.Set transmission type.Subindex = 16#02; SDO List.Set transmission type.Value = 16#FF; SDO List.Set transmission type.Size = 8; SDO List.Set transmission type.AbortIfError = FALSE; SDO List.Set transmission type.JumpToLine = FALSE; SDO List.Set transmission type.Line = 0; SDO List.Set inhibit time.Index = 16#1800; SDO List.Set inhibit time.Subindex = 16#03; SDO List.Set inhibit time.Value = 16#00C8;
              SDO List.Set inhibit time.Size = 16; SDO List.Set inhibit time.AbortIfError = FALSE; SDO List.Set inhibit time.JumpToLine = FALSE; SDO List.Set inhibit time.Line = 0; SDO List.Clear pdo mapping.Index = 16#1A00; SDO List.Clear pdo mapping.Subindex = 16#00; SDO List.Clear pdo mapping.Value = 16#0; SDO List.Clear pdo mapping.Size = 8; SDO List.Clear pdo mapping.AbortIfError = FALSE; SDO List.Clear pdo mapping.JumpToLine = FALSE; SDO List.Clear pdo mapping.Line = 0; SDO List.Set Mapping.Index = 16#1A00; SDO List.Set Mapping.Subindex = 16#01; SDO List.Set Mapping.Value = 16#21500020; SDO List.Set Mapping.Size = 32; SDO List.Set Mapping.AbortIfError = FALSE; SDO List.Set Mapping.JumpToLine = FALSE; SDO List.Set Mapping.Line = 0; SDO List.Set number of mappings.Index = 16#1A00; SDO List.Set number of mappings.Subindex = 16#00; SDO List.Set number of mappings.Value = 16#01; SDO List.Set number of mappings.Size = 8; SDO List.Set number of mappings.AbortIfError = FALSE; SDO List.Set number of mappings.JumpToLine = FALSE; SDO List.Set number of mappings.Line = 0; SDO List.Set and enable COB-ID.Index = 16#1800; SDO List.Set and enable COB-ID.Subindex = 16#01; SDO List.Set and enable COB-ID.Value = 16#000001A0; SDO List.Set and enable COB-ID.Size = 32; SDO List.Set and enable COB-ID.AbortIfError = FALSE; SDO List.Set and enable COB-ID.JumpToLine = FALSE; SDO List.Set and enable COB-ID.Line = 0; SDO List.Disable PDO.Index = 16#1801; SDO List.Disable PDO.Subindex = 16#01; SDO List.Disable PDO.Value = 16#800002A0; SDO List.Disable PDO.Size = 32; SDO List.Disable PDO.AbortIfError = FALSE; SDO List.Disable PDO.JumpToLine = FALSE; SDO List.Disable PDO.Line = 0; SDO List.Set transmission type.Index = 16#1801;
              SDO List.Set transmission type.Subindex = 16#02; SDO List.Set transmission type.Value = 16#FF; SDO List.Set transmission type.Size = 8; SDO List.Set transmission type.AbortIfError = FALSE; SDO List.Set transmission type.JumpToLine = FALSE; SDO List.Set transmission type.Line = 0; SDO List.Set inhibit time.Index = 16#1801; SDO List.Set inhibit time.Subindex = 16#03; SDO List.Set inhibit time.Value = 16#00C8; SDO List.Set inhibit time.Size = 16; SDO List.Set inhibit time.AbortIfError = FALSE; SDO List.Set inhibit time.JumpToLine = FALSE; SDO List.Set inhibit time.Line = 0; SDO List.Clear pdo mapping.Index = 16#1A01; SDO List.Clear pdo mapping.Subindex = 16#00; SDO List.Clear pdo mapping.Value = 16#0; SDO List.Clear pdo mapping.Size = 8; SDO List.Clear pdo mapping.AbortIfError = FALSE; SDO List.Clear pdo mapping.JumpToLine = FALSE; SDO List.Clear pdo mapping.Line = 0; SDO List.Set Mapping.Index = 16#1A01; SDO List.Set Mapping.Subindex = 16#01; SDO List.Set Mapping.Value = 16#220A0140; SDO List.Set Mapping.Size = 32; SDO List.Set Mapping.AbortIfError = FALSE; SDO List.Set Mapping.JumpToLine = FALSE; SDO List.Set Mapping.Line = 0; SDO List.Set number of mappings.Index = 16#1A01; SDO List.Set number of mappings.Subindex = 16#00; SDO List.Set number of mappings.Value = 16#01; SDO List.Set number of mappings.Size = 8; SDO List.Set number of mappings.AbortIfError = FALSE; SDO List.Set number of mappings.JumpToLine = FALSE; SDO List.Set number of mappings.Line = 0; SDO List.Set and enable COB-ID.Index = 16#1801; SDO List.Set and enable COB-ID.Subindex = 16#01; SDO List.Set and enable COB-ID.Value = 16#000002A0; SDO List.Set and enable COB-ID.Size = 32; SDO List.Set and enable COB-ID.AbortIfError = FALSE; SDO List.Set and enable COB-ID.JumpToLine = FALSE;
              SDO List.Set and enable COB-ID.Line = 0; SDO List.Disable PDO.Index = 16#1802; SDO List.Disable PDO.Subindex = 16#01; SDO List.Disable PDO.Value = 16#800003A0; SDO List.Disable PDO.Size = 32; SDO List.Disable PDO.AbortIfError = FALSE; SDO List.Disable PDO.JumpToLine = FALSE; SDO List.Disable PDO.Line = 0; SDO List.Set transmission type.Index = 16#1802; SDO List.Set transmission type.Subindex = 16#02; SDO List.Set transmission type.Value = 16#FF; SDO List.Set transmission type.Size = 8; SDO List.Set transmission type.AbortIfError = FALSE; SDO List.Set transmission type.JumpToLine = FALSE; SDO List.Set transmission type.Line = 0; SDO List.Set inhibit time.Index = 16#1802; SDO List.Set inhibit time.Subindex = 16#03; SDO List.Set inhibit time.Value = 16#00C8; SDO List.Set inhibit time.Size = 16; SDO List.Set inhibit time.AbortIfError = FALSE; SDO List.Set inhibit time.JumpToLine = FALSE; SDO List.Set inhibit time.Line = 0; SDO List.Clear pdo mapping.Index = 16#1A02; SDO List.Clear pdo mapping.Subindex = 16#00; SDO List.Clear pdo mapping.Value = 16#0; SDO List.Clear pdo mapping.Size = 8; SDO List.Clear pdo mapping.AbortIfError = FALSE; SDO List.Clear pdo mapping.JumpToLine = FALSE; SDO List.Clear pdo mapping.Line = 0; SDO List.Set Mapping.Index = 16#1A02; SDO List.Set Mapping.Subindex = 16#01; SDO List.Set Mapping.Value = 16#220A0240; SDO List.Set Mapping.Size = 32; SDO List.Set Mapping.AbortIfError = FALSE; SDO List.Set Mapping.JumpToLine = FALSE; SDO List.Set Mapping.Line = 0; SDO List.Set number of mappings.Index = 16#1A02; SDO List.Set number of mappings.Subindex = 16#00; SDO List.Set number of mappings.Value = 16#01; SDO List.Set number of mappings.Size = 8;
              SDO List.Set number of mappings.AbortIfError = FALSE; SDO List.Set number of mappings.JumpToLine = FALSE; SDO List.Set number of mappings.Line = 0; SDO List.Set and enable COB-ID.Index = 16#1802; SDO List.Set and enable COB-ID.Subindex = 16#01; SDO List.Set and enable COB-ID.Value = 16#000003A0; SDO List.Set and enable COB-ID.Size = 32; SDO List.Set and enable COB-ID.AbortIfError = FALSE; SDO List.Set and enable COB-ID.JumpToLine = FALSE; SDO List.Set and enable COB-ID.Line = 0; SDO List.Disable PDO.Index = 16#1803; SDO List.Disable PDO.Subindex = 16#01; SDO List.Disable PDO.Value = 16#800004A0; SDO List.Disable PDO.Size = 32; SDO List.Disable PDO.AbortIfError = FALSE; SDO List.Disable PDO.JumpToLine = FALSE; SDO List.Disable PDO.Line = 0; SDO List.Set transmission type.Index = 16#1803; SDO List.Set transmission type.Subindex = 16#02; SDO List.Set transmission type.Value = 16#FF; SDO List.Set transmission type.Size = 8; SDO List.Set transmission type.AbortIfError = FALSE; SDO List.Set transmission type.JumpToLine = FALSE; SDO List.Set transmission type.Line = 0; SDO List.Set inhibit time.Index = 16#1803; SDO List.Set inhibit time.Subindex = 16#03; SDO List.Set inhibit time.Value = 16#00C8; SDO List.Set inhibit time.Size = 16; SDO List.Set inhibit time.AbortIfError = FALSE; SDO List.Set inhibit time.JumpToLine = FALSE; SDO List.Set inhibit time.Line = 0; SDO List.Clear pdo mapping.Index = 16#1A03; SDO List.Clear pdo mapping.Subindex = 16#00; SDO List.Clear pdo mapping.Value = 16#0; SDO List.Clear pdo mapping.Size = 8; SDO List.Clear pdo mapping.AbortIfError = FALSE; SDO List.Clear pdo mapping.JumpToLine = FALSE; SDO List.Clear pdo mapping.Line = 0; SDO List.Set Mapping.Index = 16#1A03; SDO List.Set Mapping.Subindex = 16#01;
              SDO List.Set Mapping.Value = 16#220A0340; SDO List.Set Mapping.Size = 32; SDO List.Set Mapping.AbortIfError = FALSE; SDO List.Set Mapping.JumpToLine = FALSE; SDO List.Set Mapping.Line = 0; SDO List.Set number of mappings.Index = 16#1A03; SDO List.Set number of mappings.Subindex = 16#00; SDO List.Set number of mappings.Value = 16#01; SDO List.Set number of mappings.Size = 8; SDO List.Set number of mappings.AbortIfError = FALSE; SDO List.Set number of mappings.JumpToLine = FALSE; SDO List.Set number of mappings.Line = 0; SDO List.Set and enable COB-ID.Index = 16#1803; SDO List.Set and enable COB-ID.Subindex = 16#01; SDO List.Set and enable COB-ID.Value = 16#000004A0; SDO List.Set and enable COB-ID.Size = 32; SDO List.Set and enable COB-ID.AbortIfError = FALSE; SDO List.Set and enable COB-ID.JumpToLine = FALSE; SDO List.Set and enable COB-ID.Line = 0; ConfigVersion = 50659584
            unmapped channels: Write Data (mappable): Write Trigger, Write Data (mappable): Data_sub1, Write Data (mappable): Data_sub2, Write Data (mappable): Data_sub3, Device Status, Read Data (mappable): Data_sub1, Read Data (mappable): Data_sub2, Read Data (mappable): Data_sub3
*)

// Device/Application/IO
VAR_GLOBAL
	

	///////////////////////////
	// Inputs
	///////////////////////////
	
	xBG20		AT %IX1.0	: BOOL;	// Stopper released
	xBG21		AT %IX1.1	: BOOL;	// Carrier available
	xBG22		AT %IX1.2	: BOOL;	// Carrier ID bit 0
	xBG23		AT %IX1.3	: BOOL;	// Carrier ID bit 1
	xBG24		AT %IX1.4	: BOOL;	// Carrier ID bit 2
	xEmg		AT %IX0.0	: BOOL;	// Emergency stop
	
	///////////////////////////
	// Outputs
	///////////////////////////	
	
	xMB20		AT %QX1.0	: BOOL;	// Release stopper
	xQA1_LEFT	AT %QX0.5	: BOOL;	// Conveyor to the left
	xQA1_RIGHT	AT %QX0.4	: BOOL;	// Conveyor to the right
	xQA1_SLOW	AT %QX0.6	: BOOL;	// Conveyor Slow
	xQA1_STOP	AT %QX0.7	: BOOL;	// Conveyor Stop
	
	
END_VAR

// Device/Application/PLC_TO_PC_PROJECT_PRG
PROGRAM PLC_TO_PC_PROJECT_PRG
VAR
	// FLOW
	state: INT := 0;
	// RESET ITEM
	timer: TON;
	// RFID
	RFID: dc_ecp.Dtm425;
	// RFID
	rfidData: dc_ecp.st_CPF_RfidData;
	// RFID
	carrierID: UINT;
	
	// TCP
	TCPclient: dc_ecp.TcpClientByteStream;
	
	// DATE
	dtNow : DATE_AND_TIME;
	getDtNow: DTU.GetDateAndTime;
	stationID: STRING;
	dataOut: STRING(127);
	
END_VAR


CASE state OF
	
	0: //Initialization
	stationID := 'PLC_13';
	TCPclient.Connect(sIP:='172.20.66.39', uiPort:=11381);	// Connect to TCP client
	state := 100;
	
	
	100: //wait for TCP client
	IF TCPclient.xConnected AND TCPclient.xReady THEN
		state := 101;
	END_IF


	101: // Initialize RFID
	RFID.ClearError();		//Resets RFID object
	state := 102;
	
	
	102: // Wait for RFID reader to connect
	IF RFID.xReady THEN		//Check if RFID is ready and if reader is connected
		state := 103;		//Update state of program
	END_IF

	
	103: // Belt initialization
	// BASICS
	IO.xQA1_RIGHT := TRUE; 	//Starts right conveyor
	IO.xMB20 := FALSE; 		//Make sure releaser is up
	state := 104;
	

	104: // Wait for carrier to arrive
	IF IO.xBG21 = TRUE THEN //Check if carrier is available
		IO.xMB20 := TRUE; 	//Pull releaser down
		state := 200;		//Update state of program
	END_IF
	
	
	200: //Read the RFID tag
	RFID.ReadTag(uiStartAddress:=0, uiDataLength:=SIZEOF(rfidData), ADR(rfidData));	//Read data from RFID tag
	state := 201;
	
	
	201: //Wait for RFID read
	IF RFID.xReady THEN			//Check if RFID tag has been read
		carrierID := dc_ecp.SwapWORD(rfidData.uiCarrierID);
		state := 300;
	END_IF
	
	
	300: //Get date and time
	getDtNow.xExecute := TRUE;	// Execute function block to retrieve date and time
	state := 301;
	
	
	301: //Wait for date and time
	IF getDtNow.xDone THEN
		state := 302;
	END_IF
	
	
	302: //Save date and time to variable
	IF getDtNow.xDone THEN
		dtNow := getDtNow.dtDateAndTime;
		getDtNow.xExecute := FALSE;
		state := 400;
	END_IF
	
	
	400: //Assemble data to be correct format
	// Header + stationID
	dataOut := CONCAT('<plcData><stationID>',stationID);
	dataOut := CONCAT(dataOut,'</stationID>');
	
	// carrierID
	dataOut := CONCAT(dataOut,'<carrierID>');
	dataOut := CONCAT(dataOut,UINT_TO_STRING(carrierID));
	dataOut := CONCAT(dataOut,'</carrierID>');
	
	// dtNowString
	dataOut := CONCAT(dataOut,'<date>');
	dataOut := CONCAT(dataOut,DT_TO_STRING(dtNow));
	dataOut := CONCAT(dataOut,'</date>');
	
	// Footer
	dataOut := CONCAT(dataOut,'</plcData>');
	
	state := 800;
	
	
	
	
	
	
	
	
	800: // Send data using TCP/IP
	TCPclient.Send(pToSend:=ADR(dataOut), uiSizeToSend:=SIZEOF(dataOut)); // What to send and size of what is to be sent
	state := 900;
	
	
	900: // Switch belt direction
	IO.xQA1_RIGHT := FALSE; // Stop right
	IO.xMB20 := TRUE;		// Pull releaser down
	IO.xQA1_LEFT := TRUE;	// Start left
	state := 901;
	
	
	901: // Start timer
	timer(IN:=TRUE, PT:=T#5S); //Initialize timer with a 2 sec delay
	state := 902;
	
	
	902: // Wait for timer
	IF timer.Q = TRUE THEN	//Check if timer is finished
		timer(IN:=FALSE);	//Reset timer
		IO.xQA1_LEFT := FALSE;
		state := 903;			//Update state of program
	END_IF
	
	
	903: // Reset
	IO.xQA1_RIGHT := TRUE; 	// Start right
	IO.xMB20 := FALSE; 		// Pull releaser down
	state := 104;

END_CASE

TCPclient();
RFID();
timer();
getDtNow();

END_PROGRAM

// Device/Application/PLC_PRG
PROGRAM PLC_PRG
VAR
	state: UINT := 0;
END_VAR


CASE state OF
	
	0: //initialization
	IO.xQA1_RIGHT := TRUE; 	//Starts right conveyor
	IO.xMB20 := FALSE; 		//Make sure releaser is up 
	state := 1;				//Update state of program
	
	1: //wait for carrier
	IF IO.xBG21 = TRUE THEN //Check if carrier is available
		IO.xMB20 := TRUE; 	//Pull releaser down
		state := 2;			//Update state of program
	END_IF
	
	2: //Wait for the carrier to pass
	IF IO.xBG21 = FALSE THEN //Check if carrier is not there
		IO.xMB20 := FALSE;	 //Pull releaser up again
		state := 1;			 //Update state of program
	END_IF

END_CASE

END_PROGRAM

// Device/Application/RFID_PRG
PROGRAM RFID_PRG
VAR
	state: INT := 0;
	RFID: dc_ecp.Dtm425;
	rfidData: dc_ecp.st_CPF_RfidData;
	timer: TON;
	carrierID: UINT;
END_VAR


CASE state OF
	
	0: //initialization
	IO.xQA1_RIGHT := TRUE; 	//Starts right conveyor
	IO.xMB20 := FALSE; 		//Make sure releaser is up 
	RFID.ClearError();		//Resets RFID object
	state := 1;				//Update state of program
	
	1: //wait for RFID to clear
	IF RFID.xReady THEN
		RFID.Connect(usiNodeId:=32,usiNetworkId:=0,usiChannel:=1);	//Connect to RFID object		<------- PROBLEM
		state := 2;													//Update state of program
	END_IF
	
	2: //wait for RFID to connect
	IF RFID.xReady THEN	//Check if RFID is ready and if connected
		state := 3;								//Update state of program
	END_IF
	
	3: //wait for carrier
	IF IO.xBG21 = TRUE THEN //Check if carrier is available
		state := 4;			//Update state of program
	END_IF
	
	4: //Read the RFID tag
	RFID.ReadTag(uiStartAddress:=0, uiDataLength:=SIZEOF(rfidData), ADR(rfidData));	//Read data from RFID tag
	state := 5;																		//Update state
	
	5: //Wait for RFID read
	IF RFID.xReady THEN						//Check if RFID tag has been read
		carrierID := dc_ecp.SwapWORD(rfidData.uiCarrierID);
		IF carrierID <= 8 THEN				//Check ID of RFID tag
			state := 20;					//Update state according to ID
		ELSE
			state := 40;					//Update state according to ID
		END_IF
	END_IF
	
	
	20: // Release pallet 1-8
	IO.xMB20 := TRUE;	//Pull releaser down
	//IO.xQA1_SLOW := TRUE;
	state := 60;		//Update state of program
	
	40: // Release pallet 9-16
	timer(IN:=TRUE, PT:=T#10S);	//Initialize timer with 10 sec delay
	IO.xMB20 := TRUE;			//Pull releaser down
	state := 41;				//Update state
	
	41: // Wait for timer
	IF timer.Q = TRUE THEN	//Check if timer is finished
		timer(IN:=FALSE);	//Reset timer					<-----Blev ikke gjort i videoen???
		IO.xMB20 := FALSE;	//Pull releaser up
		state := 60;		//Update state
	END_IF
	
	
	
	60: // Wait for the carrier to pass
	IF IO.xBG21 = FALSE THEN //Check if carrier is not there
		IO.xMB20 := FALSE;	 //Pull releaser up again
		state := 3;			 //Update state
	END_IF
	
	

END_CASE

RFID();
timer();

END_PROGRAM

// Device/Application/timer_PRG
PROGRAM timer_PRG
VAR
	state: INT := 0;
	timer: TON;
END_VAR


CASE state OF
	
	0: //initialization
	IO.xQA1_RIGHT := TRUE; 	//Starts right conveyor
	IO.xMB20 := FALSE; 		//Make sure releaser is up 
	state := 1;				//Update state of program
	
	1: //wait for carrier
	IF IO.xBG21 = TRUE THEN //Check if carrier is available
		IO.xMB20 := TRUE; 	//Pull releaser down
		state := 2;			//Update state of program
	END_IF
	
	/////// TIMER IMPLEMENTATION ///////
	2: //activate timer
	timer(IN:=TRUE, PT:=T#2S); //Initialize timer with a 2 sec delay
	state := 3;
	
	3: //wait for timer
	IF timer.Q = TRUE THEN	//Check if timer is finished
		timer(IN:=FALSE);	//Reset timer
		IO.xMB20 := FALSE;	//Pull releaser up
		state := 1;			//Update state of program
	END_IF
	////////////////////////////////////
	
	

END_CASE

timer();

END_PROGRAM

// Device/Application/customTimer_PRG
PROGRAM customTimer_PRG
VAR
	state: INT := 0;
	timer: TON;
END_VAR


CASE state OF
	
	0: //initialization
	IO.xMB20 := FALSE; 		//Make sure releaser is up 
	state := 1;				//Update state of program
	
	1: //Move carrier right
	IO.xQA1_RIGHT := TRUE; 	//Starts conveyor moving right
	state := 2;

	2: //Wait for carrier
	IF IO.xBG21 = TRUE THEN 		//Check if carrier is available
		IO.xQA1_RIGHT := FALSE; 	//Stops conveyor moving right
		state := 3;
	END_IF

	3: //Move carrier left
	IO.xQA1_LEFT := TRUE;
	state := 4;
	
	4: //Activate timer
	timer(IN:=TRUE, PT:=T#6S); //Initialize timer with a 2 sec delay
	state := 5;
	
	5: //Wait for timer
	IF timer.Q = TRUE THEN	//Check if timer is finished
		timer(IN:=FALSE);	//Reset timer
		IO.xQA1_LEFT := FALSE;
		state := 1;			//Update state of program
	END_IF

END_CASE

timer();

END_PROGRAM

// Device/Application/TCP_PRG
PROGRAM TCP_PRG
VAR
	state: INT := 0;
	TCPclient: dc_ecp.TcpClientByteStream;
	dataOut: UINT := 69;
	dataIn: DWORD;
END_VAR


CASE state OF
	
	0: //Initialization
	IO.xQA1_RIGHT := TRUE; 	//Starts right conveyor
	IO.xMB20 := FALSE; 		//Make sure releaser is up
	TCPclient.Connect(sIP:='172.20.66.39', uiPort:=11381);
	state := 1;				//Update state of program
	
	1: //wait for TCP client
	IF TCPclient.xConnected AND TCPclient.xReady THEN
		state := 2;
	END_IF
	
	2: //Wait for carrier
	IF IO.xBG21 = TRUE THEN //Check if carrier is available
		TCPclient.Send(pToSend:=ADR(dataOut), uiSizeToSend:=SIZEOF(dataOut)); // What to send and size of what is to be sent
		state := 3;
	END_IF
	
	3: //Wait for send
	IF TCPclient.xReady THEN
		TCPclient.Receive(pToReceive:=ADR(dataIn), uiSizeToReceive:=SIZEOF(dataIn)); //What to receive and size of what is to be received
		state := 4;
	END_IF
	
	4: //Wait for receive
	IF TCPclient.xReady THEN
		//PROCESS DATA RECEIVED HERE!!!
		IO.xMB20 := TRUE; //Pull releaser down
		state := 5;
	END_IF
	
	5: //Wait for the carrier to pass
	IF IO.xBG21 = FALSE THEN //Check if carrier is not there
		IO.xMB20 := FALSE;	 //Pull releaser up again
		state := 2;			 //Update state of program				<---- He sent it to case 3
	END_IF

END_CASE

TCPclient();

END_PROGRAM
